// TIA Portal V19 export
TYPE "Prod_Beam_Ctrl"
// stored: Access Published
   STRUCT
      Setup_LinePreparation_Exe : Bool;
      STOP_FineTurno : Bool;
      STOP_ControlloQualita : Bool;
      STOP_End_Of_Production : Bool;
      Beams_Data : "Prod_Beam_Data";
   END_STRUCT;
END_TYPE
